(* Logix 5000 project; controller Sucrose_Main Emulate 5570 rev 20.12; software revision 20.01; part 23 of 30 *)
(* tags used below, declared in another part *)
   AI_E23_0 : REAL[8];   // Analog Input EN2T_FLX 192.168.1.23
   AI_E23_1 : REAL[8];   // Analog Input EN2T_FLX 192.168.1.23
   AI_E25_0 : REAL[8];   // Analog Input EN2T_FLX 192.168.1.25
   Alarm_ACK_Master_Timer : TIMER;
   DATE_TIME : Date_Time;
   DI_E23_3 : ALIAS FOR FLX_E23:3:I;   // Discrete Input EN2T_FLX 192.168.1.23
   DI_E23_4 : ALIAS FOR FLX_E23:4:I;   // Discrete Input EN2T_FLX 192.168.1.23
   DI_E25_2 : ALIAS FOR FLX_E25:2:I;   // Discrete Input EN2T_FLX 192.168.1.25
   FV230101_AOI : QSI_Flow_Valve;   // FV-23-01-01-O SUCROSE RECEIVING TO SUCROSE TANK #1 VALVE OPEN
   FV230201_AOI : QSI_Flow_Valve;   // FV-23-02-01-O SUCROSE RECEIVING TO SUCROSE TANK #2 VALVE OPEN
   FV230301_AOI : QSI_Flow_Valve;   // FV-23-03-01-O SUCROSE RECEIVING TO SUCROSE TANK #3 VALVE OPEN
   MAP_TO_SUCROSE_CIP : DINT[10];
   Messaging : Area_Ladder;
   MSG_READ_FROM_SUCROSE_CIP : MESSAGE;
   ONESHOTBITS : INT[10];
   P230010_AOI : PF525_VFD_E_ENET;   // P-23-00-10 RECEIVING PUMP 1
   P230020_AOI : PF525_VFD_E_ENET;   // P-23-00-20 RECEIVING PUMP 2
   READ_FROM_SUCROSE_CIP : DINT[10];
   Rung_Comment : BOOL;
   SucroseCIP_Drain_Inhibit : BOOL;
   SucroseCIP_FILTRATION_ALL_PATHS_Selected : BOOL;
   SucroseCIP_FILTRATION_PATH1_Selected : BOOL;
   SucroseCIP_FILTRATION_PATH2_Selected : BOOL;
   SucroseCIP_FILTRATION_PATH3_Selected : BOOL;
   SucroseCIP_FILTRATION_PATH4_Selected : BOOL;
   SucroseCIP_FILTRATION_REMOTE : CIP_REMOTE;
   SucroseCIP_HELD : BOOL;
   SucroseCIP_P230401_REMOTE : CIP_REMOTE;
   SucroseCIP_P230402_REMOTE : CIP_REMOTE;
   SucroseCIP_PAUSED : BOOL;
   SucroseCIP_Pulse_Inhibit : BOOL;
   SucroseCIP_RECEIVING2_REMOTE : CIP_REMOTE;
   SucroseCIP_RECEIVING_LINE_REMOTE : CIP_REMOTE;
   SucroseCIP_RECEIVING_REMOTE : CIP_REMOTE;
   SucroseCIP_RINGMAIN_REMOTE : CIP_REMOTE;
   SucroseCIP_RUNNING : BOOL;
   SucroseCIP_SeatLift_Pulsing : BOOL;
   SucroseCIP_TK230101_REMOTE : CIP_REMOTE;
   SucroseCIP_TK230201_REMOTE : CIP_REMOTE;
   SucroseCIP_TK230301_REMOTE : CIP_REMOTE;
   SucroseCIP_TT : BOOL;
   SucroseDischarge : Area_Program;
   SucroseFiltration : Area_Program;
   SucroseReceiving : Area_Program;
   SucroseTanks : Area_Program;
   TK_23_01_01_RECEIVING_COMPLETE : BOOL;
   TK_23_02_01_RECEIVING_COMPLETE : BOOL;
   TK_23_03_01_RECEIVING_COMPLETE : BOOL;
(* Master_Main, continued *)

ROUTINE MainRoutine   (* ladder *)
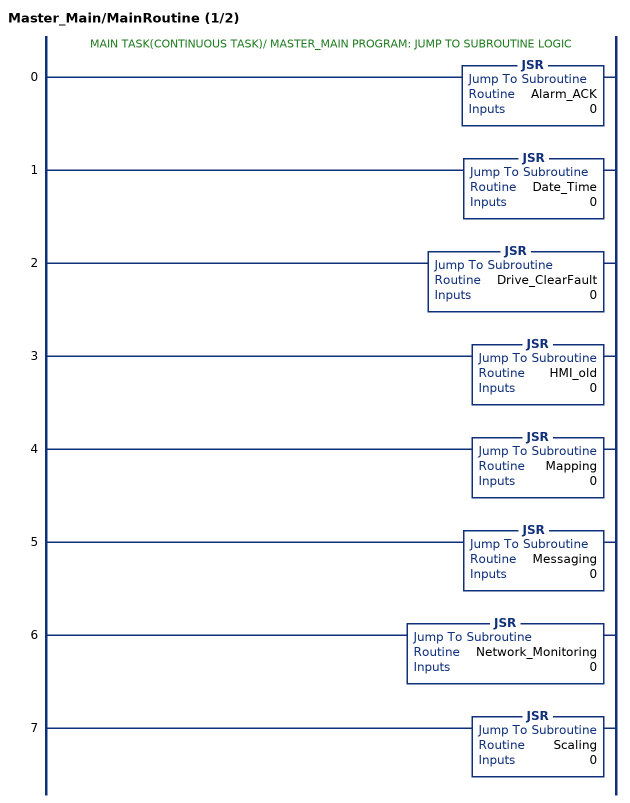
   // MAIN TASK(CONTINUOUS TASK)/ MASTER_MAIN PROGRAM: JUMP TO SUBROUTINE LOGIC
   0: JSR(Alarm_ACK,0);
   1: JSR(Date_Time,0);
   2: JSR(Drive_ClearFault,0);
   3: JSR(HMI_old,0);
   4: JSR(Mapping,0);
   5: JSR(Messaging,0);
   6: JSR(Network_Monitoring,0);
   7: JSR(Scaling,0);
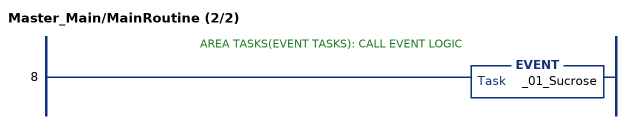
   // AREA TASKS(EVENT TASKS): CALL EVENT LOGIC
   8: EVENT(_01_Sucrose);
END_ROUTINE

ROUTINE Mapping   (* ladder *)
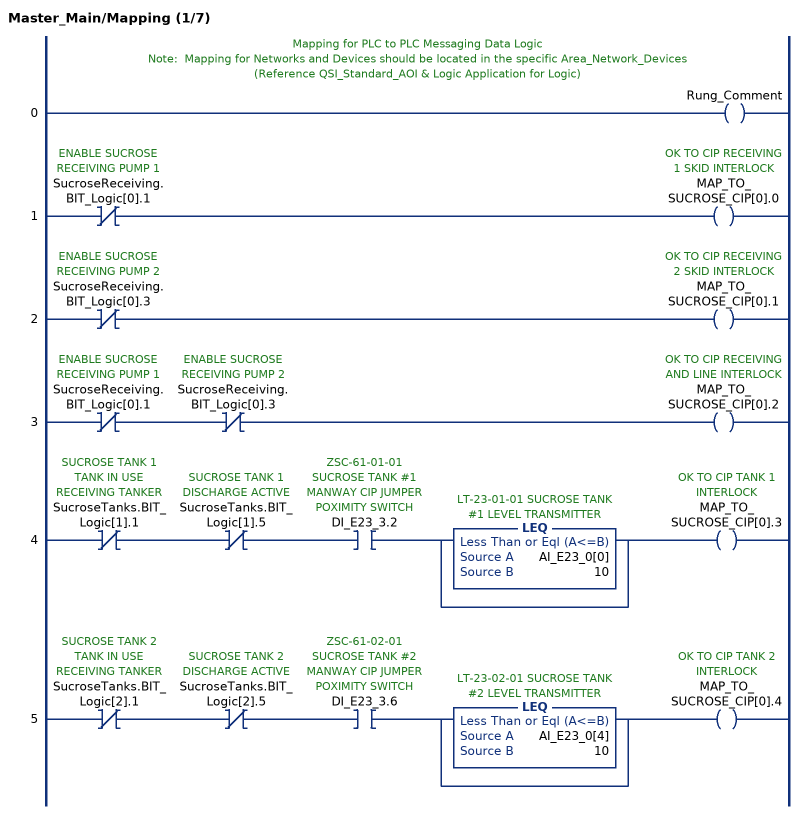
   // Mapping for PLC to PLC Messaging Data Logic
   // Note:  Mapping for Networks and Devices should be located in the specific Area_Network_Devices
   // (Reference QSI_Standard_AOI & Logic Application for Logic)
   0: OTE(Rung_Comment);
   1: XIO(SucroseReceiving.BIT_Logic[0].1)OTE(MAP_TO_SUCROSE_CIP[0].0);
   2: XIO(SucroseReceiving.BIT_Logic[0].3)OTE(MAP_TO_SUCROSE_CIP[0].1);
   3: XIO(SucroseReceiving.BIT_Logic[0].1)XIO(SucroseReceiving.BIT_Logic[0].3)OTE(MAP_TO_SUCROSE_CIP[0].2);
   4: XIO(SucroseTanks.BIT_Logic[1].1)XIO(SucroseTanks.BIT_Logic[1].5)XIC(DI_E23_3.2)[LEQ(AI_E23_0[0],10) ,]OTE(MAP_TO_SUCROSE_CIP[0].3);
   5: XIO(SucroseTanks.BIT_Logic[2].1)XIO(SucroseTanks.BIT_Logic[2].5)XIC(DI_E23_3.6)[LEQ(AI_E23_0[4],10) ,]OTE(MAP_TO_SUCROSE_CIP[0].4);
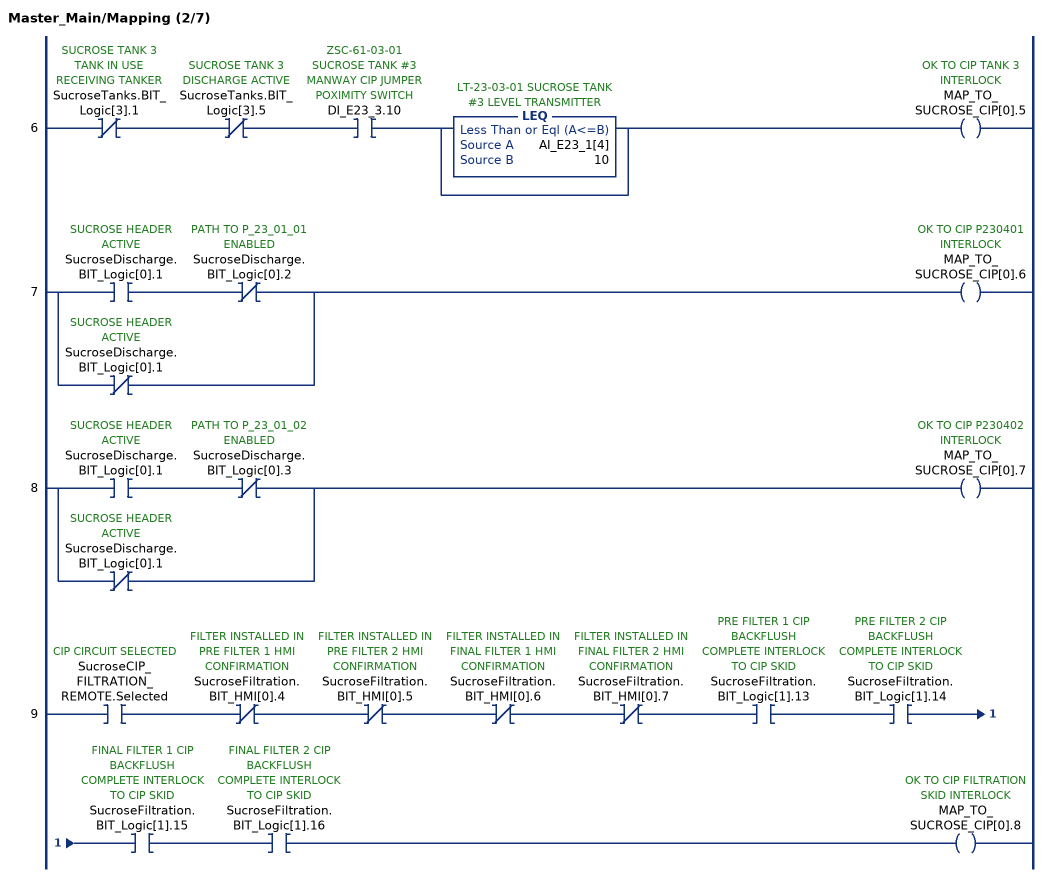
   6: XIO(SucroseTanks.BIT_Logic[3].1)XIO(SucroseTanks.BIT_Logic[3].5)XIC(DI_E23_3.10)[LEQ(AI_E23_1[4],10) ,]OTE(MAP_TO_SUCROSE_CIP[0].5);
   7: [XIC(SucroseDischarge.BIT_Logic[0].1) XIO(SucroseDischarge.BIT_Logic[0].2) ,XIO(SucroseDischarge.BIT_Logic[0].1) ]OTE(MAP_TO_SUCROSE_CIP[0].6);
   8: [XIC(SucroseDischarge.BIT_Logic[0].1) XIO(SucroseDischarge.BIT_Logic[0].3) ,XIO(SucroseDischarge.BIT_Logic[0].1) ]OTE(MAP_TO_SUCROSE_CIP[0].7);
   9: XIC(SucroseCIP_FILTRATION_REMOTE.Selected)XIO(SucroseFiltration.BIT_HMI[0].4)XIO(SucroseFiltration.BIT_HMI[0].5)XIO(SucroseFiltration.BIT_HMI[0].6)XIO(SucroseFiltration.BIT_HMI[0].7)XIC(SucroseFiltration.BIT_Logic[1].13)XIC(SucroseFiltration.BIT_Logic[1].14)XIC(SucroseFiltration.BIT_Logic[1].15)XIC(SucroseFiltration.BIT_Logic[1].16)OTE(MAP_TO_SUCROSE_CIP[0].8);
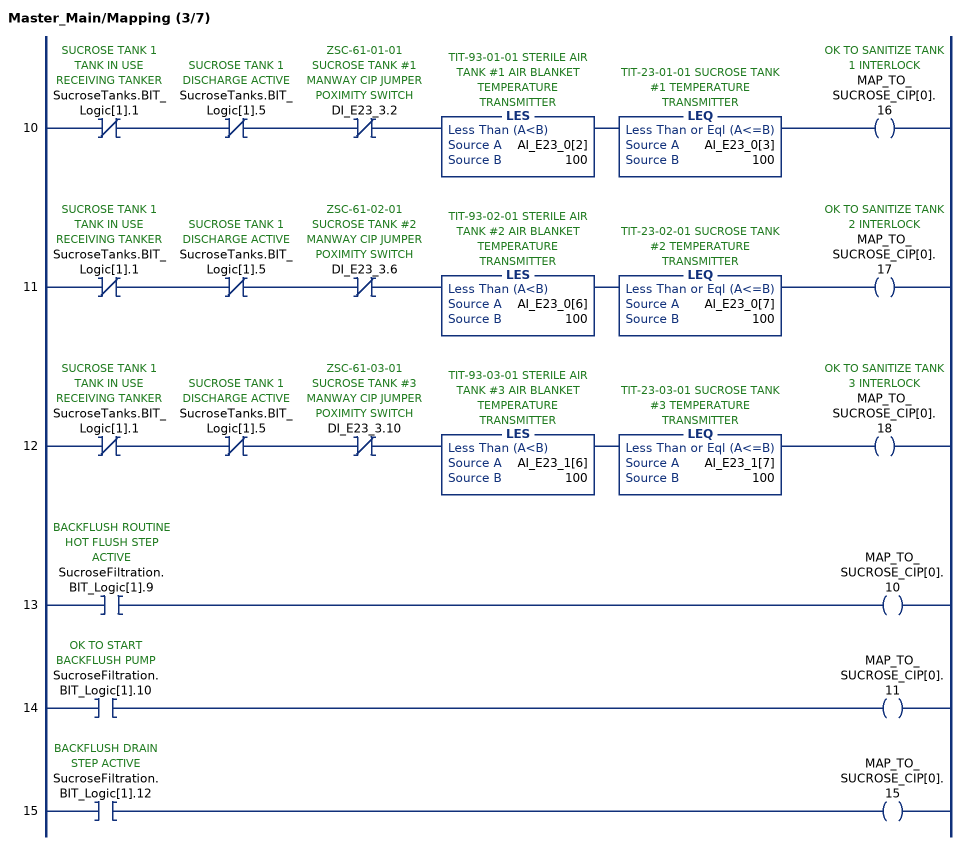
   10: XIO(SucroseTanks.BIT_Logic[1].1)XIO(SucroseTanks.BIT_Logic[1].5)XIO(DI_E23_3.2)LES(AI_E23_0[2],100)LEQ(AI_E23_0[3],100)OTE(MAP_TO_SUCROSE_CIP[0].16);
   11: XIO(SucroseTanks.BIT_Logic[1].1)XIO(SucroseTanks.BIT_Logic[1].5)XIO(DI_E23_3.6)LES(AI_E23_0[6],100)LEQ(AI_E23_0[7],100)OTE(MAP_TO_SUCROSE_CIP[0].17);
   12: XIO(SucroseTanks.BIT_Logic[1].1)XIO(SucroseTanks.BIT_Logic[1].5)XIO(DI_E23_3.10)LES(AI_E23_1[6],100)LEQ(AI_E23_1[7],100)OTE(MAP_TO_SUCROSE_CIP[0].18);
   13: XIC(SucroseFiltration.BIT_Logic[1].9)OTE(MAP_TO_SUCROSE_CIP[0].10);
   14: XIC(SucroseFiltration.BIT_Logic[1].10)OTE(MAP_TO_SUCROSE_CIP[0].11);
   15: XIC(SucroseFiltration.BIT_Logic[1].12)OTE(MAP_TO_SUCROSE_CIP[0].15);
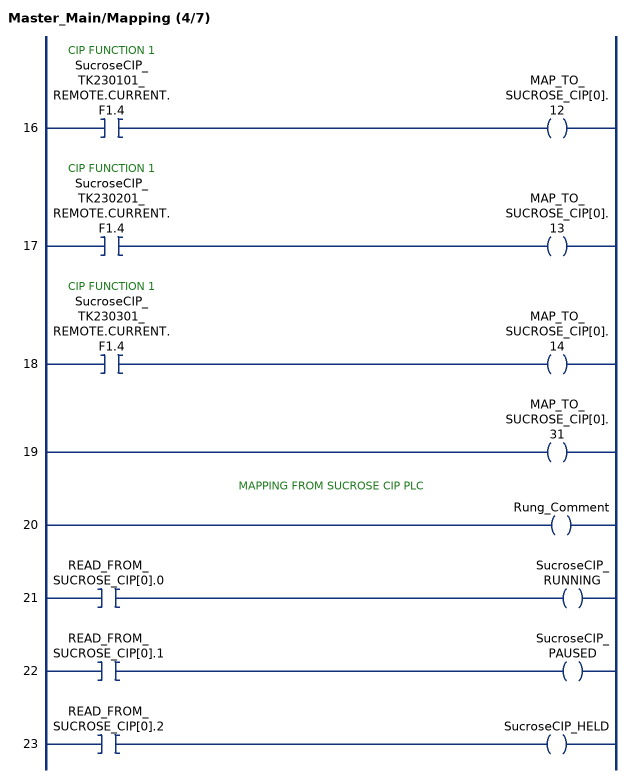
   16: XIC(SucroseCIP_TK230101_REMOTE.CURRENT.F1.4)OTE(MAP_TO_SUCROSE_CIP[0].12);
   17: XIC(SucroseCIP_TK230201_REMOTE.CURRENT.F1.4)OTE(MAP_TO_SUCROSE_CIP[0].13);
   18: XIC(SucroseCIP_TK230301_REMOTE.CURRENT.F1.4)OTE(MAP_TO_SUCROSE_CIP[0].14);
   19: OTE(MAP_TO_SUCROSE_CIP[0].31);
   // MAPPING FROM SUCROSE CIP PLC
   20: OTE(Rung_Comment);
   21: XIC(READ_FROM_SUCROSE_CIP[0].0)OTE(SucroseCIP_RUNNING);
   22: XIC(READ_FROM_SUCROSE_CIP[0].1)OTE(SucroseCIP_PAUSED);
   23: XIC(READ_FROM_SUCROSE_CIP[0].2)OTE(SucroseCIP_HELD);
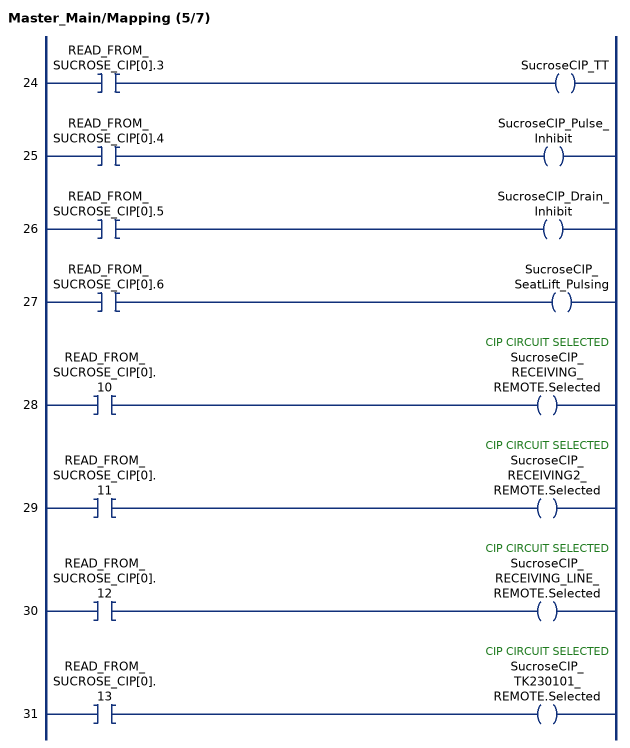
   24: XIC(READ_FROM_SUCROSE_CIP[0].3)OTE(SucroseCIP_TT);
   25: XIC(READ_FROM_SUCROSE_CIP[0].4)OTE(SucroseCIP_Pulse_Inhibit);
   26: XIC(READ_FROM_SUCROSE_CIP[0].5)OTE(SucroseCIP_Drain_Inhibit);
   27: XIC(READ_FROM_SUCROSE_CIP[0].6)OTE(SucroseCIP_SeatLift_Pulsing);
   28: XIC(READ_FROM_SUCROSE_CIP[0].10)OTE(SucroseCIP_RECEIVING_REMOTE.Selected);
   29: XIC(READ_FROM_SUCROSE_CIP[0].11)OTE(SucroseCIP_RECEIVING2_REMOTE.Selected);
   30: XIC(READ_FROM_SUCROSE_CIP[0].12)OTE(SucroseCIP_RECEIVING_LINE_REMOTE.Selected);
   31: XIC(READ_FROM_SUCROSE_CIP[0].13)OTE(SucroseCIP_TK230101_REMOTE.Selected);
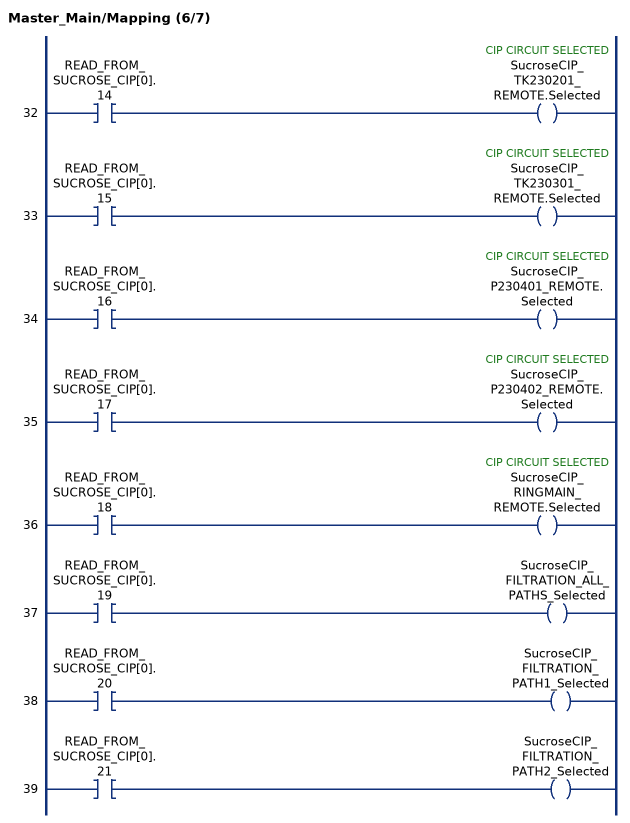
   32: XIC(READ_FROM_SUCROSE_CIP[0].14)OTE(SucroseCIP_TK230201_REMOTE.Selected);
   33: XIC(READ_FROM_SUCROSE_CIP[0].15)OTE(SucroseCIP_TK230301_REMOTE.Selected);
   34: XIC(READ_FROM_SUCROSE_CIP[0].16)OTE(SucroseCIP_P230401_REMOTE.Selected);
   35: XIC(READ_FROM_SUCROSE_CIP[0].17)OTE(SucroseCIP_P230402_REMOTE.Selected);
   36: XIC(READ_FROM_SUCROSE_CIP[0].18)OTE(SucroseCIP_RINGMAIN_REMOTE.Selected);
   37: XIC(READ_FROM_SUCROSE_CIP[0].19)OTE(SucroseCIP_FILTRATION_ALL_PATHS_Selected);
   38: XIC(READ_FROM_SUCROSE_CIP[0].20)OTE(SucroseCIP_FILTRATION_PATH1_Selected);
   39: XIC(READ_FROM_SUCROSE_CIP[0].21)OTE(SucroseCIP_FILTRATION_PATH2_Selected);
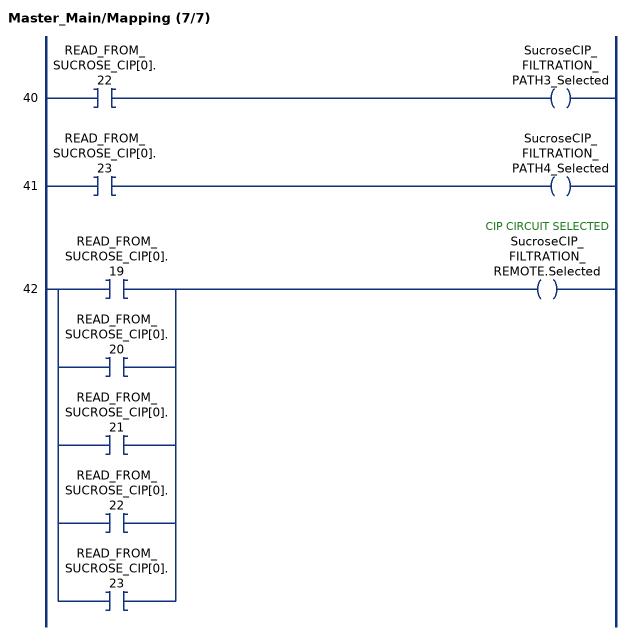
   40: XIC(READ_FROM_SUCROSE_CIP[0].22)OTE(SucroseCIP_FILTRATION_PATH3_Selected);
   41: XIC(READ_FROM_SUCROSE_CIP[0].23)OTE(SucroseCIP_FILTRATION_PATH4_Selected);
   42: [XIC(READ_FROM_SUCROSE_CIP[0].19) ,XIC(READ_FROM_SUCROSE_CIP[0].20) ,XIC(READ_FROM_SUCROSE_CIP[0].21) ,XIC(READ_FROM_SUCROSE_CIP[0].22) ,XIC(READ_FROM_SUCROSE_CIP[0].23) ]OTE(SucroseCIP_FILTRATION_REMOTE.Selected);
END_ROUTINE

ROUTINE Messaging   (* ladder *)
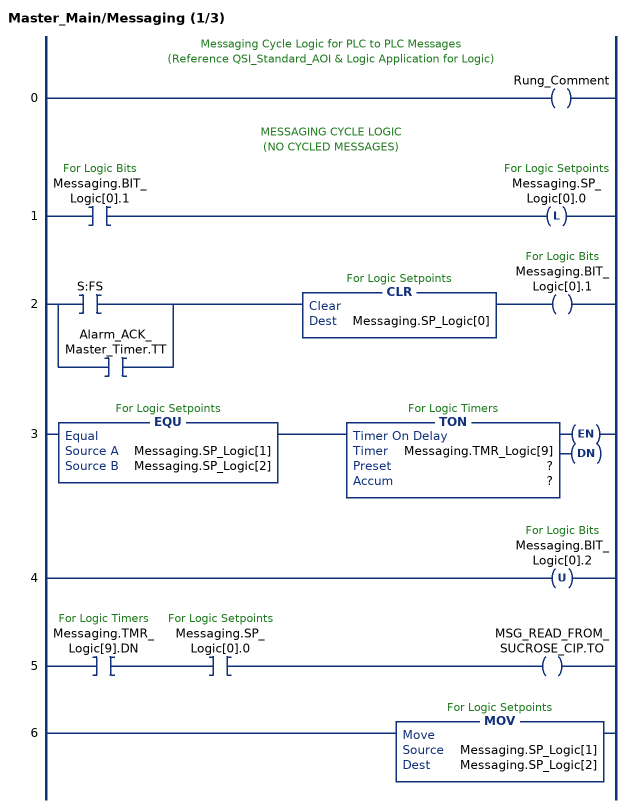
   // Messaging Cycle Logic for PLC to PLC Messages
   // (Reference QSI_Standard_AOI & Logic Application for Logic)
   0: OTE(Rung_Comment);
   // MESSAGING CYCLE LOGIC
   // (NO CYCLED MESSAGES)
   1: XIC(Messaging.BIT_Logic[0].1)OTL(Messaging.SP_Logic[0].0);
   2: [XIC(S:FS) ,XIC(Alarm_ACK_Master_Timer.TT) ]CLR(Messaging.SP_Logic[0])OTE(Messaging.BIT_Logic[0].1);
   3: EQU(Messaging.SP_Logic[1],Messaging.SP_Logic[2])TON(Messaging.TMR_Logic[9],?,?);
   4: OTU(Messaging.BIT_Logic[0].2);
   5: XIC(Messaging.TMR_Logic[9].DN)XIC(Messaging.SP_Logic[0].0)OTE(MSG_READ_FROM_SUCROSE_CIP.TO);
   6: MOV(Messaging.SP_Logic[1],Messaging.SP_Logic[2]);
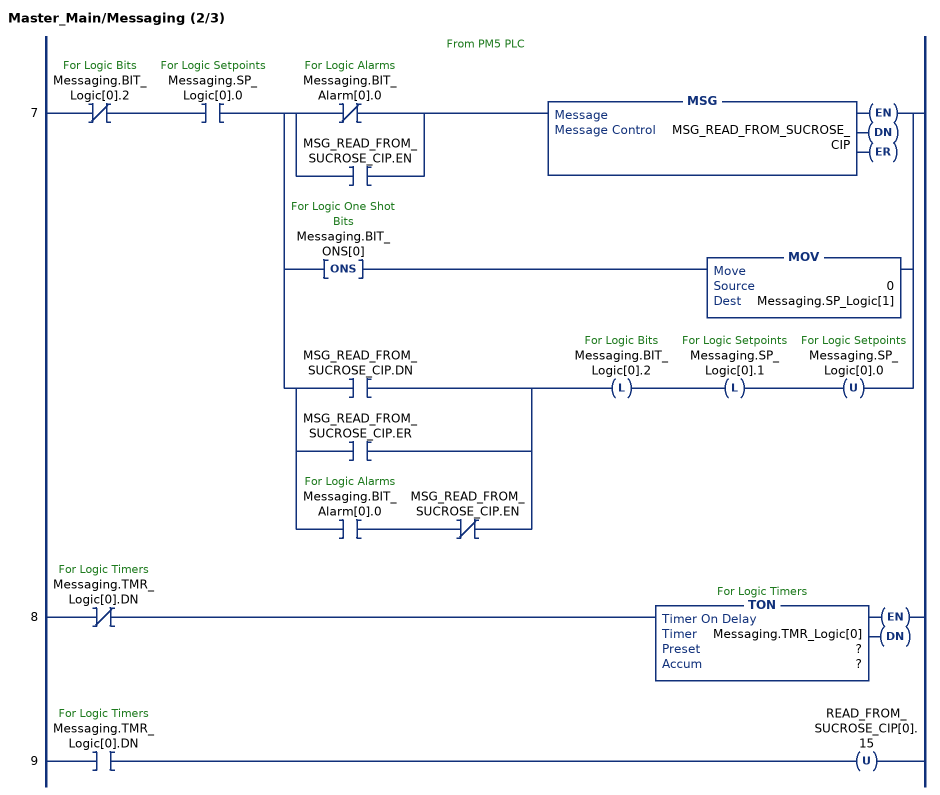
   // From PM5 PLC
   7: XIO(Messaging.BIT_Logic[0].2)XIC(Messaging.SP_Logic[0].0)[[XIO(Messaging.BIT_Alarm[0].0) ,XIC(MSG_READ_FROM_SUCROSE_CIP.EN) ] MSG(MSG_READ_FROM_SUCROSE_CIP) ,ONS(Messaging.BIT_ONS[0]) MOV(0,Messaging.SP_Logic[1]) ,[XIC(MSG_READ_FROM_SUCROSE_CIP.DN) ,XIC(MSG_READ_FROM_SUCROSE_CIP.ER) ,XIC(Messaging.BIT_Alarm[0].0) XIO(MSG_READ_FROM_SUCROSE_CIP.EN) ] OTL(Messaging.BIT_Logic[0].2) OTL(Messaging.SP_Logic[0].1) OTU(Messaging.SP_Logic[0].0) ];
   8: XIO(Messaging.TMR_Logic[0].DN)TON(Messaging.TMR_Logic[0],?,?);
   9: XIC(Messaging.TMR_Logic[0].DN)OTU(READ_FROM_SUCROSE_CIP[0].15);
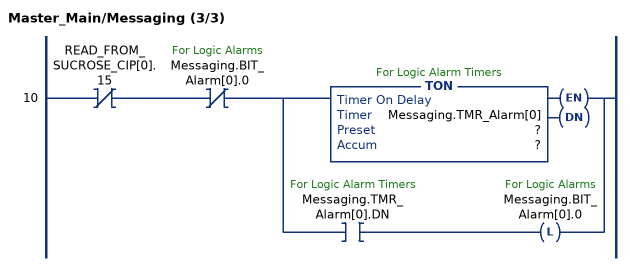
   10: XIO(READ_FROM_SUCROSE_CIP[0].15)XIO(Messaging.BIT_Alarm[0].0)[TON(Messaging.TMR_Alarm[0],?,?) ,XIC(Messaging.TMR_Alarm[0].DN) OTL(Messaging.BIT_Alarm[0].0) ];
END_ROUTINE

ROUTINE Network_Monitoring   (* ladder *)
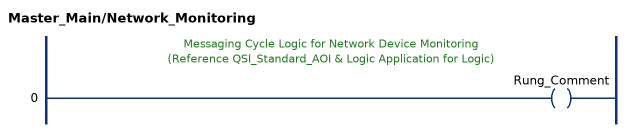
   // Messaging Cycle Logic for Network Device Monitoring
   // (Reference QSI_Standard_AOI & Logic Application for Logic)
   0: OTE(Rung_Comment);
END_ROUTINE

ROUTINE Scaling   (* ladder *)
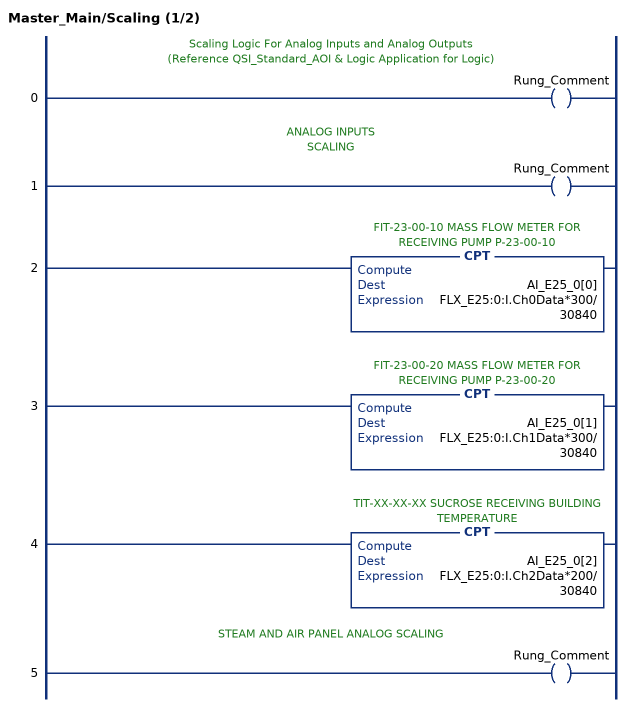
   // Scaling Logic For Analog Inputs and Analog Outputs
   // (Reference QSI_Standard_AOI & Logic Application for Logic)
   0: OTE(Rung_Comment);
   // ANALOG INPUTS
   // SCALING
   1: OTE(Rung_Comment);
   2: CPT(AI_E25_0[0],FLX_E25:0:I.Ch0Data*300/30840);
   3: CPT(AI_E25_0[1],FLX_E25:0:I.Ch1Data*300/30840);
   4: CPT(AI_E25_0[2],FLX_E25:0:I.Ch2Data*200/30840);
   // STEAM AND AIR PANEL ANALOG SCALING
   5: OTE(Rung_Comment);
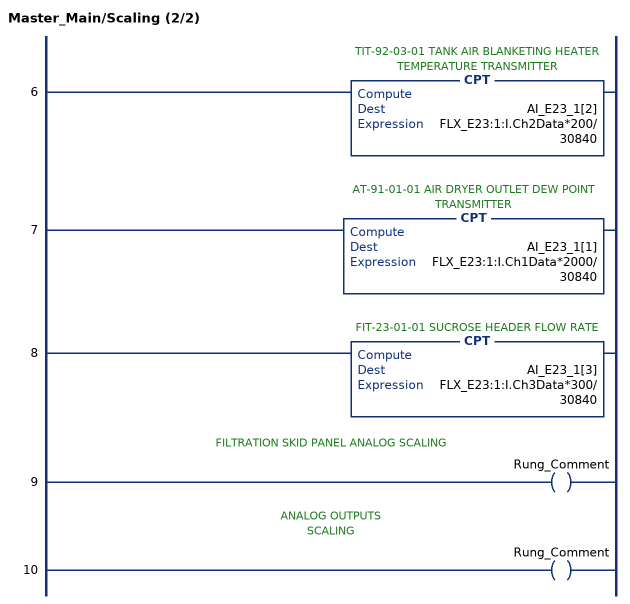
   6: CPT(AI_E23_1[2],FLX_E23:1:I.Ch2Data*200/30840);
   7: CPT(AI_E23_1[1],FLX_E23:1:I.Ch1Data*2000/30840);
   8: CPT(AI_E23_1[3],FLX_E23:1:I.Ch3Data*300/30840);
   // FILTRATION SKID PANEL ANALOG SCALING
   9: OTE(Rung_Comment);
   // ANALOG OUTPUTS
   // SCALING
   10: OTE(Rung_Comment);
END_ROUTINE
END_PROGRAM

PROGRAM ReceivingArea_AutoLogic   (* main routine MainRoutine *)

ROUTINE Alarm_Logic   (* ladder *)
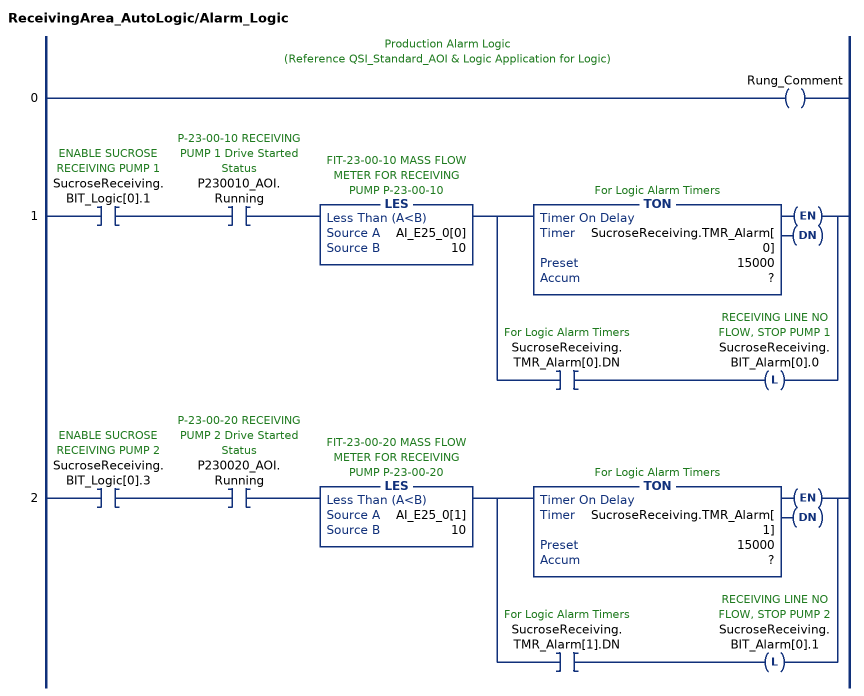
   // Production Alarm Logic
   // (Reference QSI_Standard_AOI & Logic Application for Logic)
   0: OTE(Rung_Comment);
   1: XIC(SucroseReceiving.BIT_Logic[0].1)XIC(P230010_AOI.Running)LES(AI_E25_0[0],10)[TON(SucroseReceiving.TMR_Alarm[0],?,?) ,XIC(SucroseReceiving.TMR_Alarm[0].DN) OTL(SucroseReceiving.BIT_Alarm[0].0) ];
   2: XIC(SucroseReceiving.BIT_Logic[0].3)XIC(P230020_AOI.Running)LES(AI_E25_0[1],10)[TON(SucroseReceiving.TMR_Alarm[1],?,?) ,XIC(SucroseReceiving.TMR_Alarm[1].DN) OTL(SucroseReceiving.BIT_Alarm[0].1) ];
END_ROUTINE

ROUTINE Control_Logic   (* ladder *)
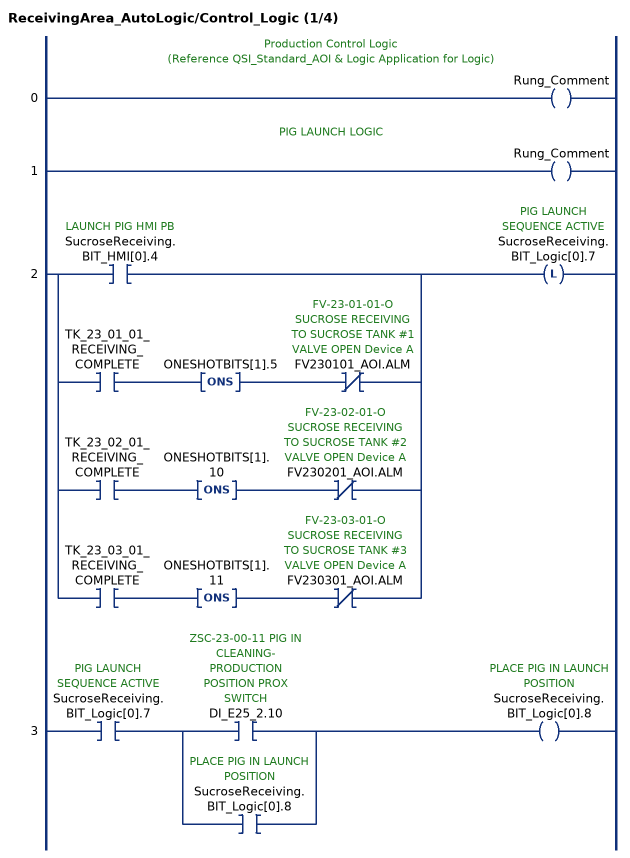
   // Production Control Logic
   // (Reference QSI_Standard_AOI & Logic Application for Logic)
   0: OTE(Rung_Comment);
   // PIG LAUNCH LOGIC
   1: OTE(Rung_Comment);
   2: [XIC(SucroseReceiving.BIT_HMI[0].4) ,XIC(TK_23_01_01_RECEIVING_COMPLETE) ONS(ONESHOTBITS[1].5) XIO(FV230101_AOI.ALM) ,XIC(TK_23_02_01_RECEIVING_COMPLETE) ONS(ONESHOTBITS[1].10) XIO(FV230201_AOI.ALM) ,XIC(TK_23_03_01_RECEIVING_COMPLETE) ONS(ONESHOTBITS[1].11) XIO(FV230301_AOI.ALM) ]OTL(SucroseReceiving.BIT_Logic[0].7);
   3: XIC(SucroseReceiving.BIT_Logic[0].7)[XIC(DI_E25_2.10) ,XIC(SucroseReceiving.BIT_Logic[0].8) ]OTE(SucroseReceiving.BIT_Logic[0].8);
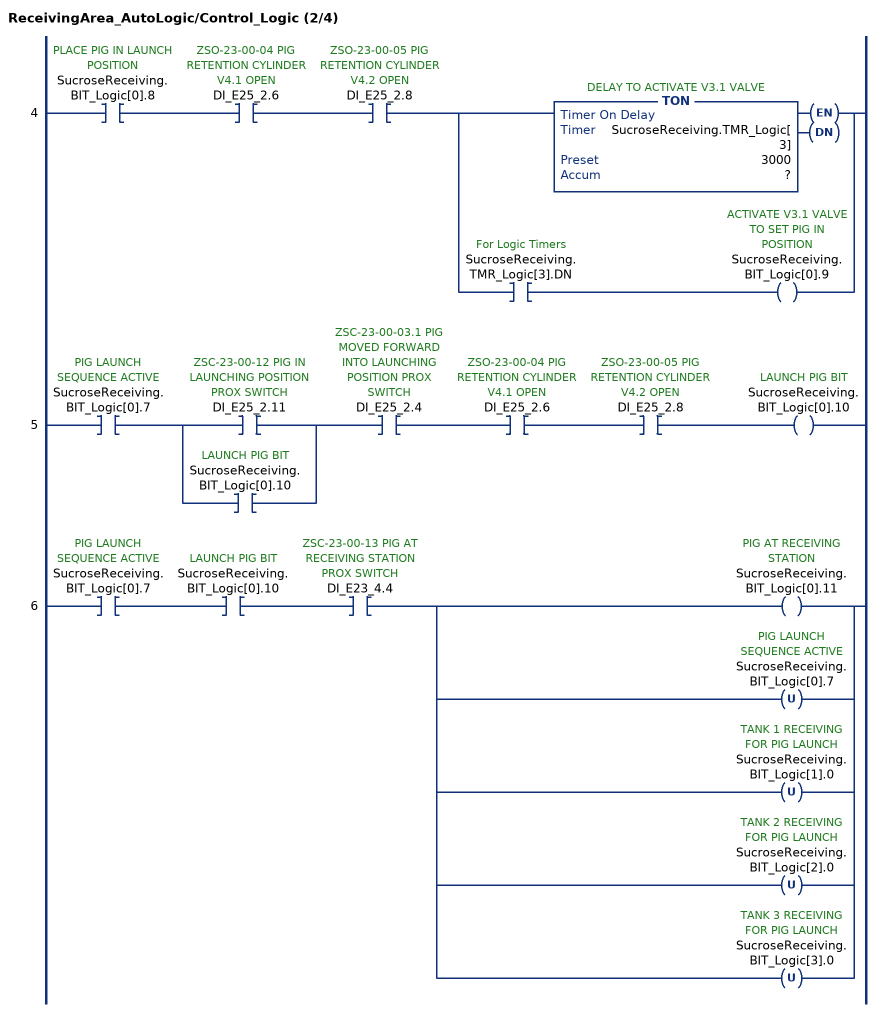
   4: XIC(SucroseReceiving.BIT_Logic[0].8)XIC(DI_E25_2.6)XIC(DI_E25_2.8)[TON(SucroseReceiving.TMR_Logic[3],?,?) ,XIC(SucroseReceiving.TMR_Logic[3].DN) OTE(SucroseReceiving.BIT_Logic[0].9) ];
   5: XIC(SucroseReceiving.BIT_Logic[0].7)[XIC(DI_E25_2.11) ,XIC(SucroseReceiving.BIT_Logic[0].10) ]XIC(DI_E25_2.4)XIC(DI_E25_2.6)XIC(DI_E25_2.8)OTE(SucroseReceiving.BIT_Logic[0].10);
   6: XIC(SucroseReceiving.BIT_Logic[0].7)XIC(SucroseReceiving.BIT_Logic[0].10)XIC(DI_E23_4.4)[OTE(SucroseReceiving.BIT_Logic[0].11) ,OTU(SucroseReceiving.BIT_Logic[0].7) ,OTU(SucroseReceiving.BIT_Logic[1].0) ,OTU(SucroseReceiving.BIT_Logic[2].0) ,OTU(SucroseReceiving.BIT_Logic[3].0) ];
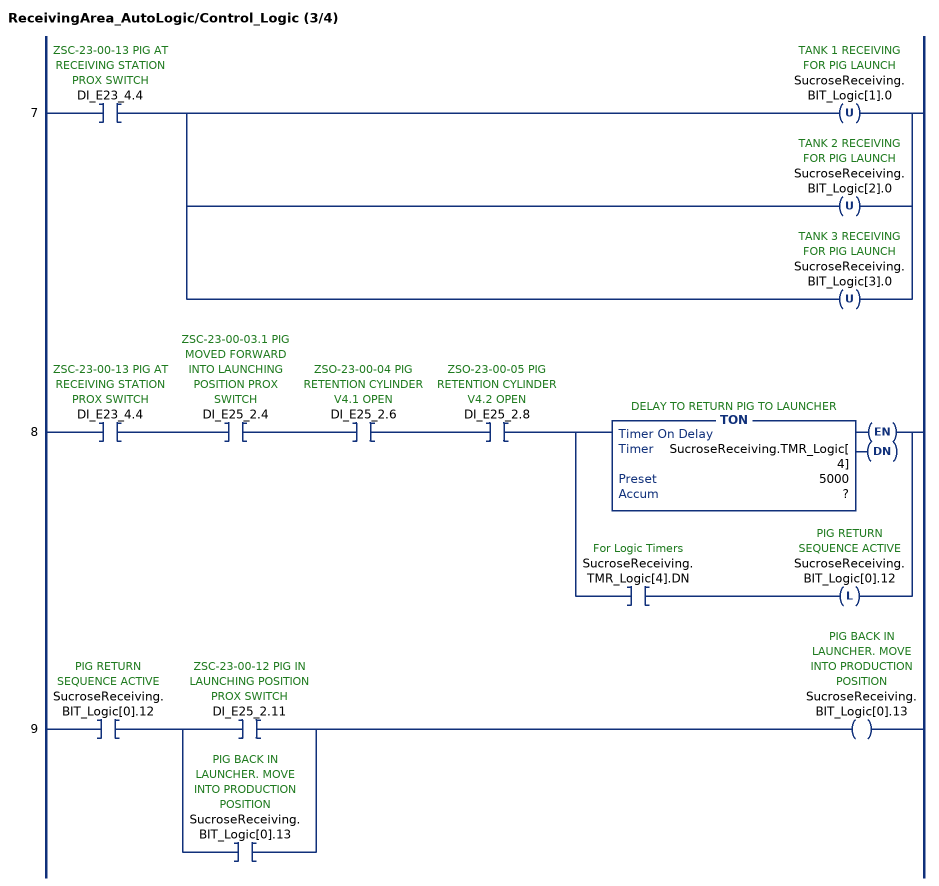
   7: XIC(DI_E23_4.4)[OTU(SucroseReceiving.BIT_Logic[1].0) ,OTU(SucroseReceiving.BIT_Logic[2].0) ,OTU(SucroseReceiving.BIT_Logic[3].0) ];
   8: XIC(DI_E23_4.4)XIC(DI_E25_2.4)XIC(DI_E25_2.6)XIC(DI_E25_2.8)[TON(SucroseReceiving.TMR_Logic[4],?,?) ,XIC(SucroseReceiving.TMR_Logic[4].DN) OTL(SucroseReceiving.BIT_Logic[0].12) ];
   9: XIC(SucroseReceiving.BIT_Logic[0].12)[XIC(DI_E25_2.11) ,XIC(SucroseReceiving.BIT_Logic[0].13) ]OTE(SucroseReceiving.BIT_Logic[0].13);
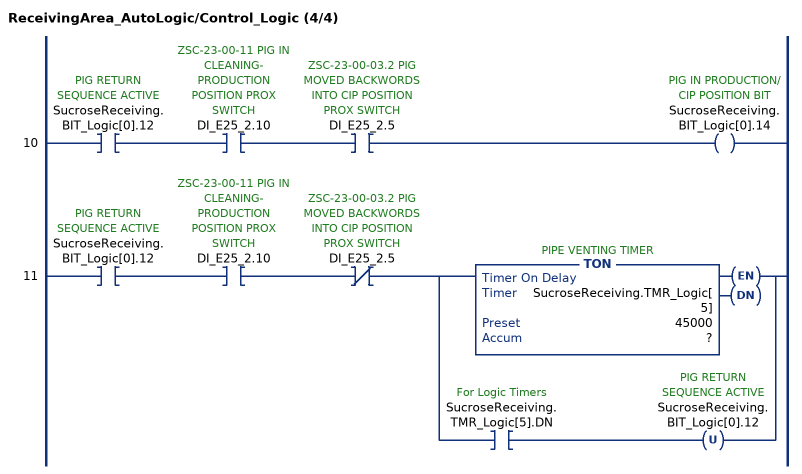
   10: XIC(SucroseReceiving.BIT_Logic[0].12)XIC(DI_E25_2.10)XIC(DI_E25_2.5)OTE(SucroseReceiving.BIT_Logic[0].14);
   11: XIC(SucroseReceiving.BIT_Logic[0].12)XIC(DI_E25_2.10)XIO(DI_E25_2.5)[TON(SucroseReceiving.TMR_Logic[5],?,?) ,XIC(SucroseReceiving.TMR_Logic[5].DN) OTU(SucroseReceiving.BIT_Logic[0].12) ];
END_ROUTINE
